(* IEC 61131-3 sources: statemachine/src/Deprecated, 4 files *)

(* ---- StateStatus.st ---- *)
NAMESPACE Simatic.Ax.StatePattern

    // Legacy runtime status structure used by the deprecated state context.
    TYPE StateStatus :
        STRUCT
            isRunning : Bool;
            activeTime : TIME;
            remainingTime : LTIME;
        END_STRUCT;
    END_TYPE

END_NAMESPACE

(* ---- IState.st ---- *)
NAMESPACE Simatic.Ax.StatePattern
    INTERFACE IState
        // Executes the active state in the deprecated state pattern.
        METHOD Execute
            VAR_INPUT
                context : REF_TO StateContext;
            END_VAR
        END_METHOD

        // Called when the deprecated context enters the state.
        METHOD OnEntry
            VAR_INPUT
                context : REF_TO StateContext;
            END_VAR
        END_METHOD

        // Called when the deprecated context leaves the state.
        METHOD OnExit
            VAR_INPUT
                context : REF_TO StateContext;
            END_VAR
        END_METHOD

        // Called when the deprecated timeout expires.
        METHOD OnTimeout
            VAR_INPUT
                context : REF_TO StateContext;
            END_VAR
        END_METHOD

    END_INTERFACE
END_NAMESPACE

(* ---- BaseState.st ---- *)
USING Simatic.Ax.StatePattern;
NAMESPACE Simatic.Ax.StatePattern
    // Legacy base state from the deprecated state pattern implementation.
    CLASS StateBase IMPLEMENTS IState
        VAR
            _nextState : IState;
            _nextStateTimeout : IState;
        END_VAR

        METHOD PUBLIC Config
            VAR_INPUT
                nextState : IState;
                nextStateTimeout : IState;
            END_VAR
            // Stores the normal and timeout successor states.
            _nextState := nextState;
            _nextStateTimeout := nextStateTimeout;
        END_METHOD

        METHOD PUBLIC OnTimeout
            VAR_INPUT
                context : REF_TO StateContext;
            END_VAR
            // Deprecated default implementation intentionally does nothing.
            ;
        END_METHOD

        METHOD PUBLIC Execute
            VAR_INPUT
                context : REF_TO StateContext;
            END_VAR
            // Deprecated default implementation intentionally does nothing.
            ;
        END_METHOD

        METHOD PUBLIC OnEntry
            VAR_INPUT
                context : REF_TO StateContext;
            END_VAR;
            // Deprecated default implementation intentionally does nothing.
        END_METHOD

        METHOD PUBLIC OnExit
            VAR_INPUT
                context : REF_TO StateContext;
            END_VAR;
            // Deprecated default implementation intentionally does nothing.
        END_METHOD

    END_CLASS
END_NAMESPACE

(* ---- StateContext.st ---- *)
USING System.Timer;

NAMESPACE Simatic.Ax.StatePattern
    // Legacy controller from the deprecated state pattern implementation.
    CLASS PUBLIC StateContext
        VAR PUBLIC

        END_VAR
        VAR
            _count : INT;
            _state : IState;
            _ton : OnDelay;
            _first : BOOL;
            _status : StateStatus;
        END_VAR

        METHOD PUBLIC InitialState : BOOL
            VAR_INPUT
                newState : IState;
                timeout : TIME;
                reset : BOOL;
            END_VAR

            // The initial state is only applied once unless reset is requested explicitly.
            IF (newState <> NULL) THEN
                IF (NOT _first OR reset) THEN
                    THIS.setState(newState := newState, timeout := timeout);
                    _first := TRUE;
                END_IF;
                InitialState := TRUE;
            ELSE
                InitialState := FALSE;
            END_IF;

        END_METHOD

        METHOD PUBLIC FINAL SetState
            VAR_INPUT
                newState : IState;
                timeout : TIME;
            END_VAR

            // Before switching states, the current state receives OnExit.
            IF (_state <> NULL) THEN
                _state.OnExit(context := REF(THIS));
            END_IF;

            IF (newState <> NULL) THEN
                _state := newState;
                _status.isRunning := TRUE;

                // The new state is entered once immediately after activation.
                _state.onEntry(context := REF(THIS));

                // A positive timeout arms the legacy TON instance.
                IF (timeout > T#0ms) THEN
                    _ton.duration := timeout;
                    _ton.signal := TRUE;
                END_IF;
                _state.Execute(context := REF(THIS));

            END_IF;
        END_METHOD

        METHOD PUBLIC FINAL Execute
            // No execution happens until an initial state has been configured.
            IF (_state = NULL) THEN
                RETURN;
            END_IF;
            _count := _count + 1;
            _ton();

            // Timeout handling is evaluated before the regular Execute call.
            IF (_ton.output) THEN
                _ton.signal := FALSE;
                _ton();
                _status.remainingTime := _ton.elapsedTime;
                _state.OnTimeout(context := REF(THIS));
            END_IF;

            _state.Execute(context := REF(THIS));
        END_METHOD

    END_CLASS
END_NAMESPACE
